// Mitsubishi GX Works2 project: Automation_EX2)   PLC: FX3G

// global labels: Global1
VAR_GLOBAL
  Start AT X007 : BOOL;
  Emergency AT X005 : BOOL;
  InventoryCheck AT M11 : BOOL;
  Valid AT M10 : BOOL;
  ReadyForWork AT Y007 : BOOL;
  IceCream AT X001 : BOOL;
  OpeningInventoryRaspberry AT D1100 : REAL;
  CurentInventoryRaspberry AT D1102 : REAL;
  OpeningInventoryLemon AT D1104 : REAL;
  CurentInventoryLemon AT D1106 : REAL;
  OpeningInventoryStabilizer AT D1108 : REAL;
  CurentInventoryStabilizer AT D1110 : REAL;
  OpeningInventoryGumy AT D1112 : REAL;
  CurentInventoryGumy AT D1114 : REAL;
  AnalogicInput AT D8280 : INT;
END_VAR
VAR_GLOBAL CONSTANT
  small5 : INT := 5;
  Big6 : INT := 6;
  Rgular : INT;
  Rgular5 : INT := 5;
  Rgular0 : INT;
  Treat6 : INT := 6;
  Treat10 : INT := 10;
END_VAR
VAR_GLOBAL
  Select_Regular AT M21 : BOOL;
  Select_Treat AT M31 : BOOL;
  SystemActive AT X007 : BOOL;
  Regular_Selected AT M100 : BOOL;
  Treat_Selected AT M200 : BOOL;
  Working_Lamp AT Y000 : BOOL;
  TC_5 AT TC5 : BOOL;
  Timer5_Done AT TS5 : BOOL;
END_VAR
VAR_GLOBAL CONSTANT
  Const_RR : REAL;
  Const_385 : REAL := 385.0;
  Const_210 : REAL := 210.0;
  Const_665 : REAL := 665.0;
  Const_70 : REAL := 70.0;
  Const_280 : REAL := 280.0;
  Const_105 : REAL := 105.0;
  Const_28 : REAL := 28.0;
  Const_455 : REAL := 455.0;
  Const_50 : INT := K50;
END_VAR
VAR_GLOBAL
  Timer5 AT TC50 : BOOL;
  CON50 AT K50 : INT;
  TC5 AT TC5 : BOOL;
  Timerrr AT TC5 : BOOL;
  Timer2 AT TC6 : BOOL;
  Timer2_done AT TS6 : BOOL;
  Shake AT X002 : BOOL;
  Cooling AT X002 : BOOL;
  Temp AT X003 : BOOL;
  CoolingTimer AT TC80 : BOOL;
  CON_80 AT K80 : INT;
  StageOneFinished AT M300 : BOOL;
  TempLowerThen10 AT X003 : BOOL;
  CoolTimerStop AT TC3 : BOOL;
  CoolTimerStoped AT TS80 : BOOL;
  CoolingLamp AT Y002 : BOOL;
  ReadyForShake AT M350 : BOOL;
END_VAR
VAR_GLOBAL CONSTANT
  Const280 : REAL := 280.0;
  Const_490 : REAL := 490.0;
END_VAR
VAR_GLOBAL
  LemonMakingTank AT D1116 : REAL;
  RaspberyMakingTank AT D1118 : REAL;
END_VAR
VAR_GLOBAL CONSTANT
  Const_350 : REAL := 350.0;
  Const_560 : REAL := 560.0;
  Const_700 : REAL := 700.0;
END_VAR
VAR_GLOBAL
  LemonCoolingTank AT D1120 : REAL;
  RaspberyCoolingTank AT D1122 : REAL;
  ShakingTank AT D1124 : REAL;
END_VAR
VAR_GLOBAL CONSTANT
  Const_1 : REAL := 1;
END_VAR
VAR_GLOBAL
  XXXXX AT M500 : BOOL;
  XXXXxx AT M500 : BOOL;
  Start_Mixing AT M500 : BOOL;
  Con30 AT K30 : INT;
  Mixing_Lamp AT TC30 : BOOL;
  Mixing_Reg_Lamp AT TC30 : BOOL;
  Mixing_Trt_Lamp AT TC50 : BOOL;
  Mixing_Done AT M501 : BOOL;
  Un_Timer AT TC21 : BOOL;
  Timer20 AT TS20 : BOOL;
  Timer21 AT TS21 : BOOL;
  Timer_20 AT TC20 : BOOL;
  Mixing_Lamp1 AT Y005 : BOOL;
  Mixing_Lamp2 AT Y006 : BOOL;
  Total_Packages AT D5000 : INT;
  M50Mixing_Done1 AT M501 : BOOL;
END_VAR
VAR_GLOBAL CONSTANT
  Rgular2000 : INT := 2000;
  Treat2400 : INT := 2400;
  Treat4000 : INT := 4000;
END_VAR
VAR_GLOBAL
  InventoryCheck12 AT M12 : BOOL;
  InventoryCheck13 AT M13 : BOOL;
  InventoryCheck14 AT M14 : BOOL;
  InventoryCheck15 AT M15 : BOOL;
  InventoryCheck16 AT M16 : BOOL;
  InventoryCheck17 AT M17 : BOOL;
  InventoryCheck18 AT M18 : BOOL;
  InventoryCheck19 AT M19 : BOOL;
  ReadyForShake1 AT M350 : BOOL;
  Start_Mixing1 AT M360 : BOOL;
  Mixing_Done1 AT M370 : BOOL;
  Station_Pack1 AT D5002 : REAL;
  Const10 AT E10 : REAL;
  Const_0 AT K0 : INT;
  Const_40 AT E40 : REAL;
  AnalogOutput AT D8282 : INT;
  Sensor_Error_Lamp AT Y011 : BOOL;
  Special_Relay AT M8013 : BOOL;
  Blink_Counter AT CS0 : BOOL;
  Const_5 AT K5 : INT;
  Analog_In_Error AT M380 : BOOL;
END_VAR
VAR_GLOBAL CONSTANT
  Treat4030 : INT := 4030;
  Rgular2030 : INT := 2030;
END_VAR
VAR_GLOBAL
  Low_Range_Regular AT M20 : BOOL;
  Low_Range_Treat AT M30 : BOOL;
END_VAR

// task Task_01 (event TRUE, interval 0, priority 31): POU_01

PROGRAM POU_01
(* structured ladder/FBD written out as ST: instructions are called as NAME(EN, inputs, outputs); _pN, _eN, _tN stand for wires *)
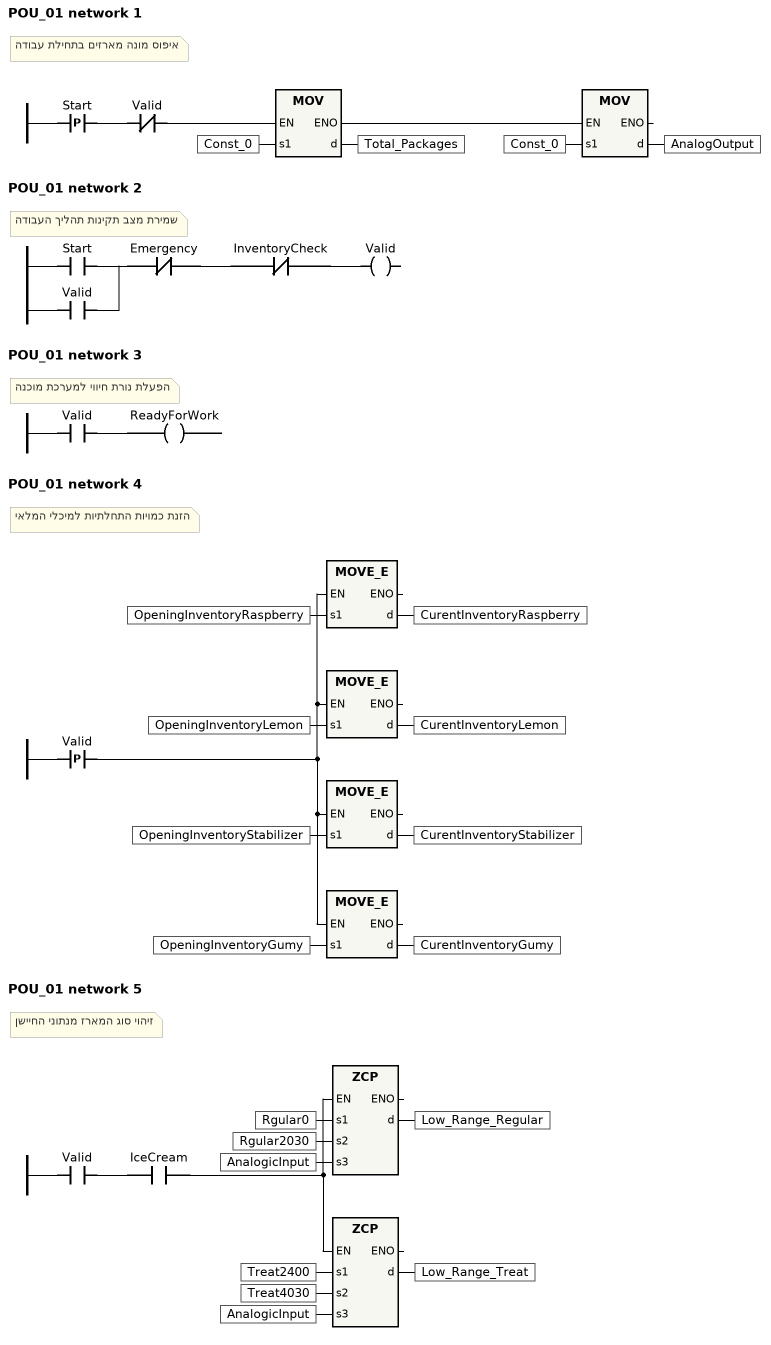
(* network 1 *)
(* איפוס מונה מארזים בתחילת עבודה *)
_e1 := MOV(LDP(TRUE, Start) AND NOT Valid, Const_0, Total_Packages);
MOV(_e1, Const_0, AnalogOutput);
(* network 2 *)
(* שמירת מצב תקינות תהליך העבודה *)
Valid := ((Start OR Valid) AND NOT Emergency) AND NOT InventoryCheck;
(* network 3 *)
(* הפעלת נורת חיווי למערכת מוכנה *)
ReadyForWork := Valid;
(* network 4 *)
(* הזנת כמויות התחלתיות למיכלי המלאי *)
_p1 := LDP(TRUE, Valid);
MOVE_E(_p1, OpeningInventoryRaspberry, CurentInventoryRaspberry);
MOVE_E(_p1, OpeningInventoryLemon, CurentInventoryLemon);
MOVE_E(_p1, OpeningInventoryStabilizer, CurentInventoryStabilizer);
MOVE_E(_p1, OpeningInventoryGumy, CurentInventoryGumy);
(* network 5 *)
(* זיהוי סוג המארז מנתוני החיישן *)
_p1 := Valid AND IceCream;
ZCP(_p1, Rgular0, Rgular2030, AnalogicInput, Low_Range_Regular);
ZCP(_p1, Treat2400, Treat4030, AnalogicInput, Low_Range_Treat);
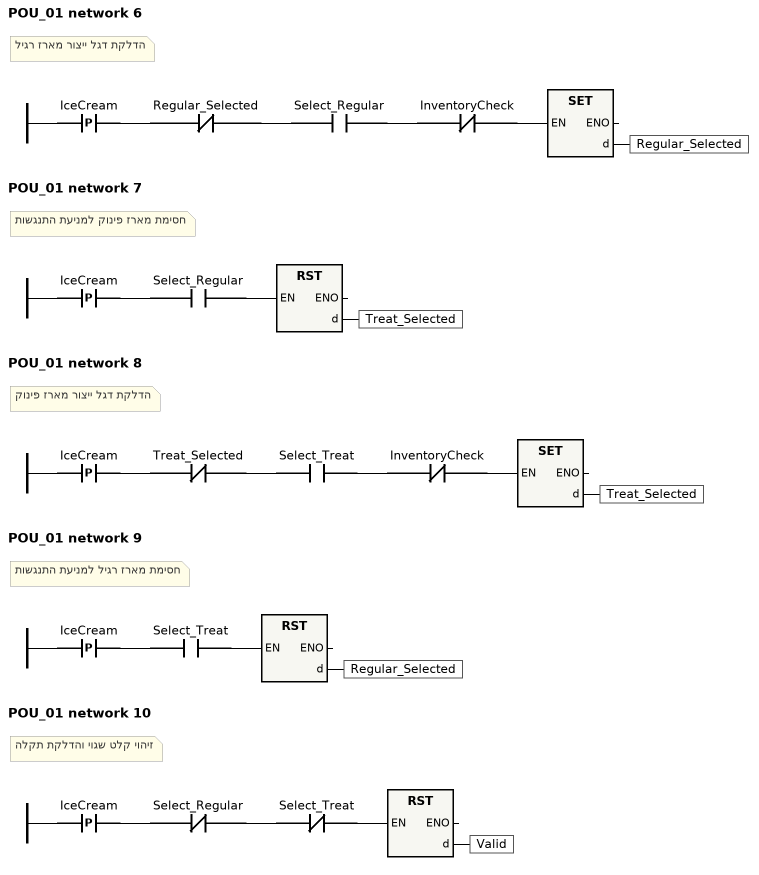
(* network 6 *)
(* הדלקת דגל ייצור מארז רגיל *)
SET(LDP(TRUE, IceCream) AND NOT Regular_Selected AND Select_Regular AND NOT InventoryCheck, Regular_Selected);
(* network 7 *)
(* חסימת מארז פינוק למניעת התנגשות *)
RST(LDP(TRUE, IceCream) AND Select_Regular, Treat_Selected);
(* network 8 *)
(* הדלקת דגל ייצור מארז פינוק *)
SET(LDP(TRUE, IceCream) AND NOT Treat_Selected AND Select_Treat AND NOT InventoryCheck, Treat_Selected);
(* network 9 *)
(* חסימת מארז רגיל למניעת התנגשות *)
RST(LDP(TRUE, IceCream) AND Select_Treat, Regular_Selected);
(* network 10 *)
(* זיהוי קלט שגוי והדלקת תקלה *)
RST(LDP(TRUE, IceCream) AND NOT Select_Regular AND NOT Select_Treat, Valid);
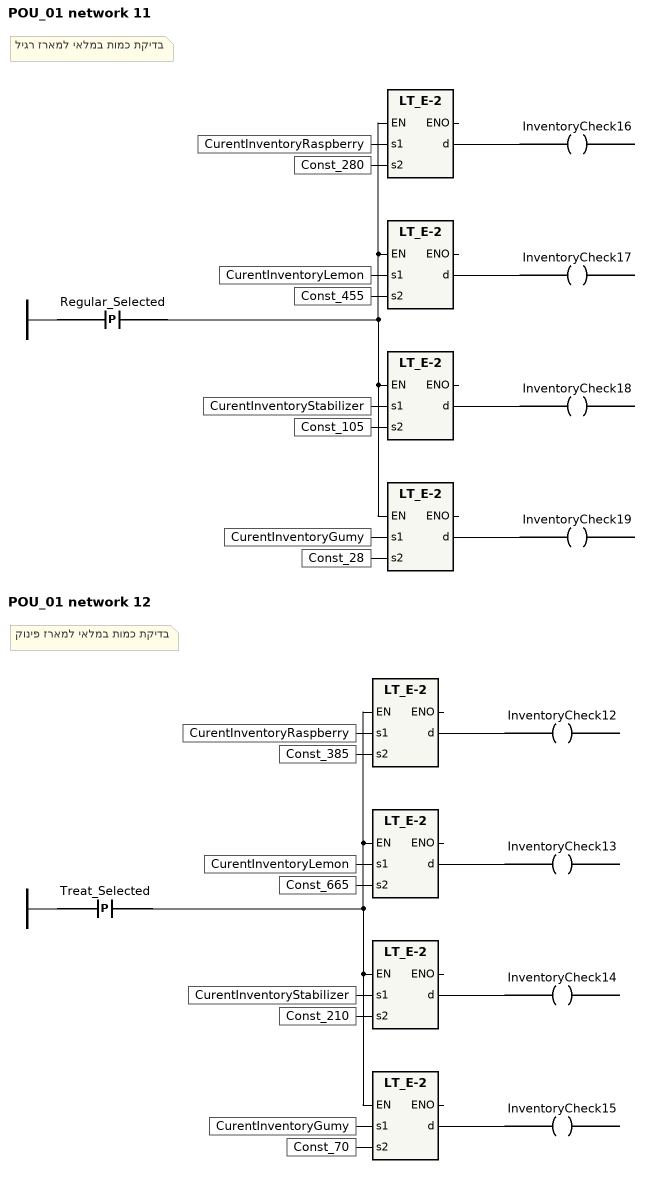
(* network 11 *)
(* בדיקת כמות במלאי למארז רגיל *)
_p1 := LDP(TRUE, Regular_Selected);
LT_E(_p1, CurentInventoryRaspberry, Const_280, _t2);
InventoryCheck16 := _t2;
LT_E(_p1, CurentInventoryLemon, Const_455, _t3);
InventoryCheck17 := _t3;
LT_E(_p1, CurentInventoryStabilizer, Const_105, _t4);
InventoryCheck18 := _t4;
LT_E(_p1, CurentInventoryGumy, Const_28, _t5);
InventoryCheck19 := _t5;
(* network 12 *)
(* בדיקת כמות במלאי למארז פינוק *)
_p1 := LDP(TRUE, Treat_Selected);
LT_E(_p1, CurentInventoryRaspberry, Const_385, _t2);
InventoryCheck12 := _t2;
LT_E(_p1, CurentInventoryLemon, Const_665, _t3);
InventoryCheck13 := _t3;
LT_E(_p1, CurentInventoryStabilizer, Const_210, _t4);
InventoryCheck14 := _t4;
LT_E(_p1, CurentInventoryGumy, Const_70, _t5);
InventoryCheck15 := _t5;
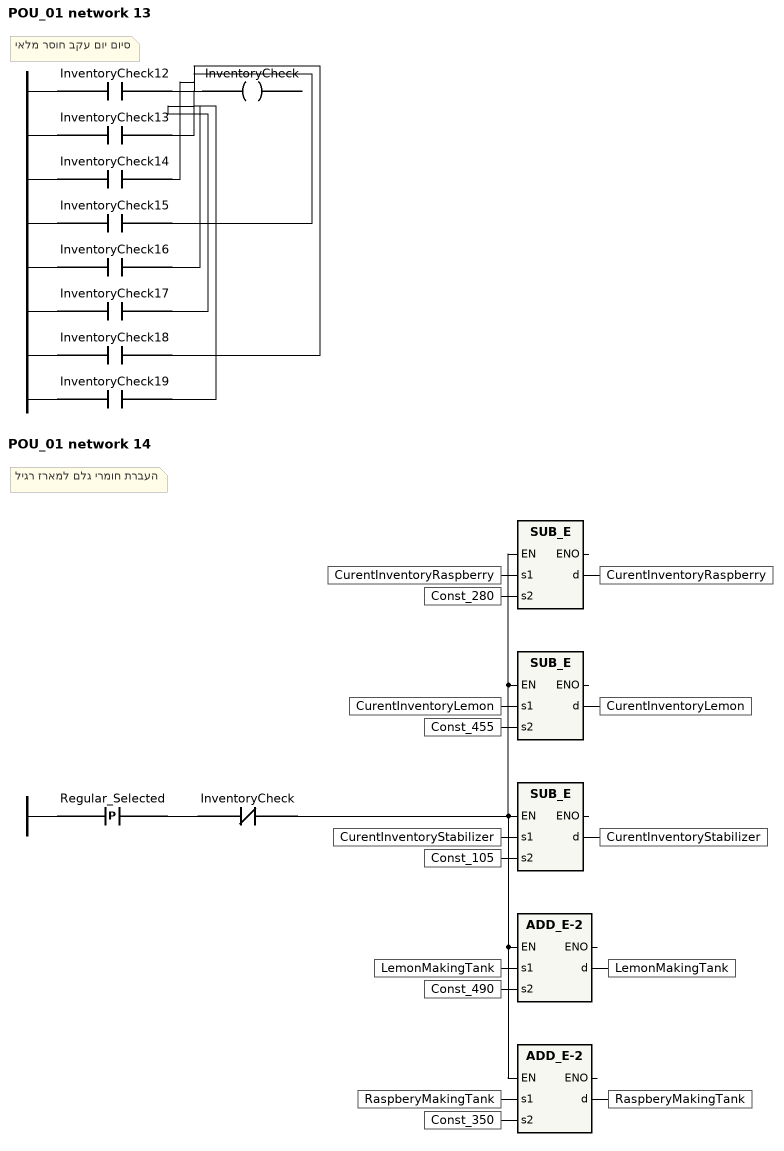
(* network 13 *)
(* סיום יום עקב חוסר מלאי *)
InventoryCheck := InventoryCheck12 OR InventoryCheck13 OR InventoryCheck14 OR InventoryCheck15 OR InventoryCheck16 OR InventoryCheck17 OR InventoryCheck18 OR InventoryCheck19;
(* network 14 *)
(* העברת חומרי גלם למארז רגיל *)
_p1 := LDP(TRUE, Regular_Selected) AND NOT InventoryCheck;
SUB_E(_p1, CurentInventoryRaspberry, Const_280, CurentInventoryRaspberry);
SUB_E(_p1, CurentInventoryLemon, Const_455, CurentInventoryLemon);
SUB_E(_p1, CurentInventoryStabilizer, Const_105, CurentInventoryStabilizer);
ADD_E(_p1, LemonMakingTank, Const_490, LemonMakingTank);
ADD_E(_p1, RaspberyMakingTank, Const_350, RaspberyMakingTank);
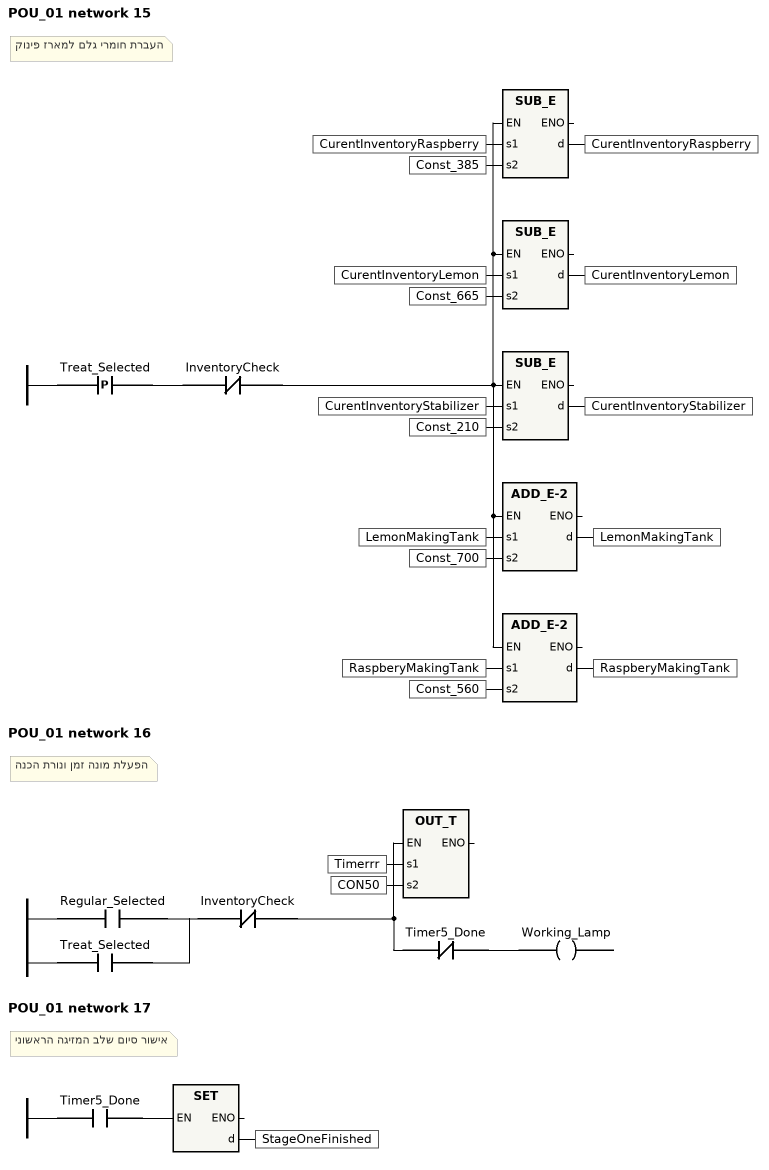
(* network 15 *)
(* העברת חומרי גלם למארז פינוק *)
_p1 := LDP(TRUE, Treat_Selected) AND NOT InventoryCheck;
SUB_E(_p1, CurentInventoryRaspberry, Const_385, CurentInventoryRaspberry);
SUB_E(_p1, CurentInventoryLemon, Const_665, CurentInventoryLemon);
SUB_E(_p1, CurentInventoryStabilizer, Const_210, CurentInventoryStabilizer);
ADD_E(_p1, LemonMakingTank, Const_700, LemonMakingTank);
ADD_E(_p1, RaspberyMakingTank, Const_560, RaspberyMakingTank);
(* network 16 *)
(* הפעלת מונה זמן ונורת הכנה *)
_p1 := (Regular_Selected OR Treat_Selected) AND NOT InventoryCheck;
OUT_T(_p1, Timerrr, CON50);
Working_Lamp := _p1 AND NOT Timer5_Done;
(* network 17 *)
(* אישור סיום שלב המזיגה הראשוני *)
SET(Timer5_Done, StageOneFinished);
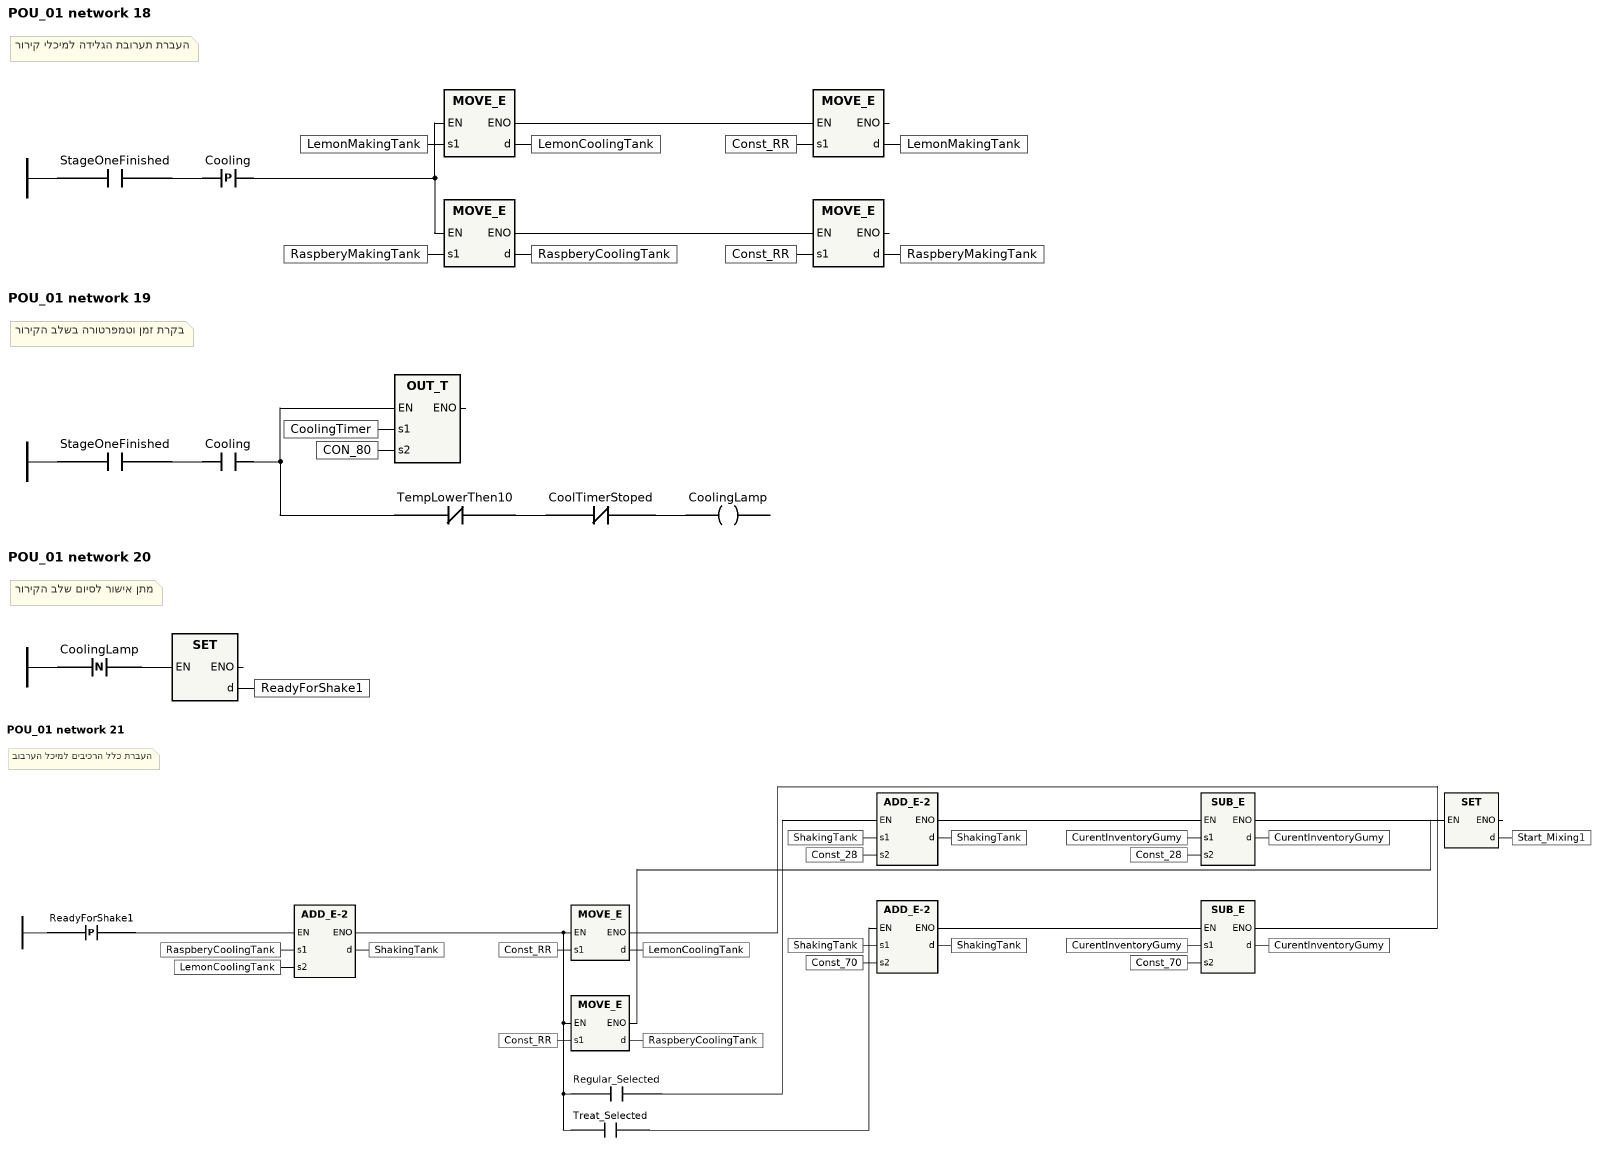
(* network 18 *)
(* העברת תערובת הגלידה למיכלי קירור *)
_p1 := StageOneFinished AND LDP(TRUE, Cooling);
_e2 := MOVE_E(_p1, LemonMakingTank, LemonCoolingTank);
MOVE_E(_e2, Const_RR, LemonMakingTank);
_e3 := MOVE_E(_p1, RaspberyMakingTank, RaspberyCoolingTank);
MOVE_E(_e3, Const_RR, RaspberyMakingTank);
(* network 19 *)
(* בקרת זמן וטמפרטורה בשלב הקירור *)
_p1 := StageOneFinished AND Cooling;
OUT_T(_p1, CoolingTimer, CON_80);
CoolingLamp := _p1 AND NOT TempLowerThen10 AND NOT CoolTimerStoped;
(* network 20 *)
(* מתן אישור לסיום שלב הקירור *)
SET(LDF(TRUE, CoolingLamp), ReadyForShake1);
(* network 21 *)
(* העברת כלל הרכיבים למיכל הערבוב *)
_e1 := ADD_E(LDP(TRUE, ReadyForShake1), RaspberyCoolingTank, LemonCoolingTank, ShakingTank);
_e2 := ADD_E(_e1 AND Regular_Selected, ShakingTank, Const_28, ShakingTank);
_e3 := SUB_E(_e2, CurentInventoryGumy, Const_28, CurentInventoryGumy);
_e4 := ADD_E(_e1 AND Treat_Selected, ShakingTank, Const_70, ShakingTank);
_e5 := SUB_E(_e4, CurentInventoryGumy, Const_70, CurentInventoryGumy);
_e6 := MOVE_E(_e1, Const_RR, LemonCoolingTank);
_e7 := MOVE_E(_e1, Const_RR, RaspberyCoolingTank);
SET(_e3 OR _e5 OR _e6 OR _e7, Start_Mixing1);
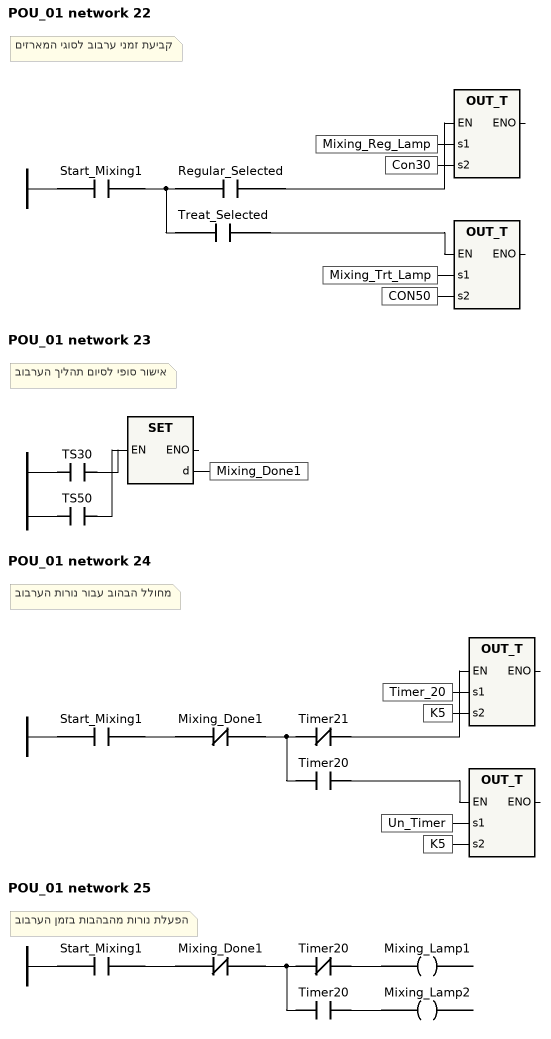
(* network 22 *)
(* קביעת זמני ערבוב לסוגי המארזים *)
OUT_T(Start_Mixing1 AND Regular_Selected, Mixing_Reg_Lamp, Con30);
OUT_T(Start_Mixing1 AND Treat_Selected, Mixing_Trt_Lamp, CON50);
(* network 23 *)
(* אישור סופי לסיום תהליך הערבוב *)
SET(TS30 OR TS50, Mixing_Done1);
(* network 24 *)
(* מחולל הבהוב עבור נורות הערבוב *)
_p1 := Start_Mixing1 AND NOT Mixing_Done1;
OUT_T(_p1 AND NOT Timer21, Timer_20, K5);
OUT_T(_p1 AND Timer20, Un_Timer, K5);
(* network 25 *)
(* הפעלת נורות מהבהבות בזמן הערבוב *)
_p1 := Start_Mixing1 AND NOT Mixing_Done1;
Mixing_Lamp1 := _p1 AND NOT Timer20;
Mixing_Lamp2 := _p1 AND Timer20;
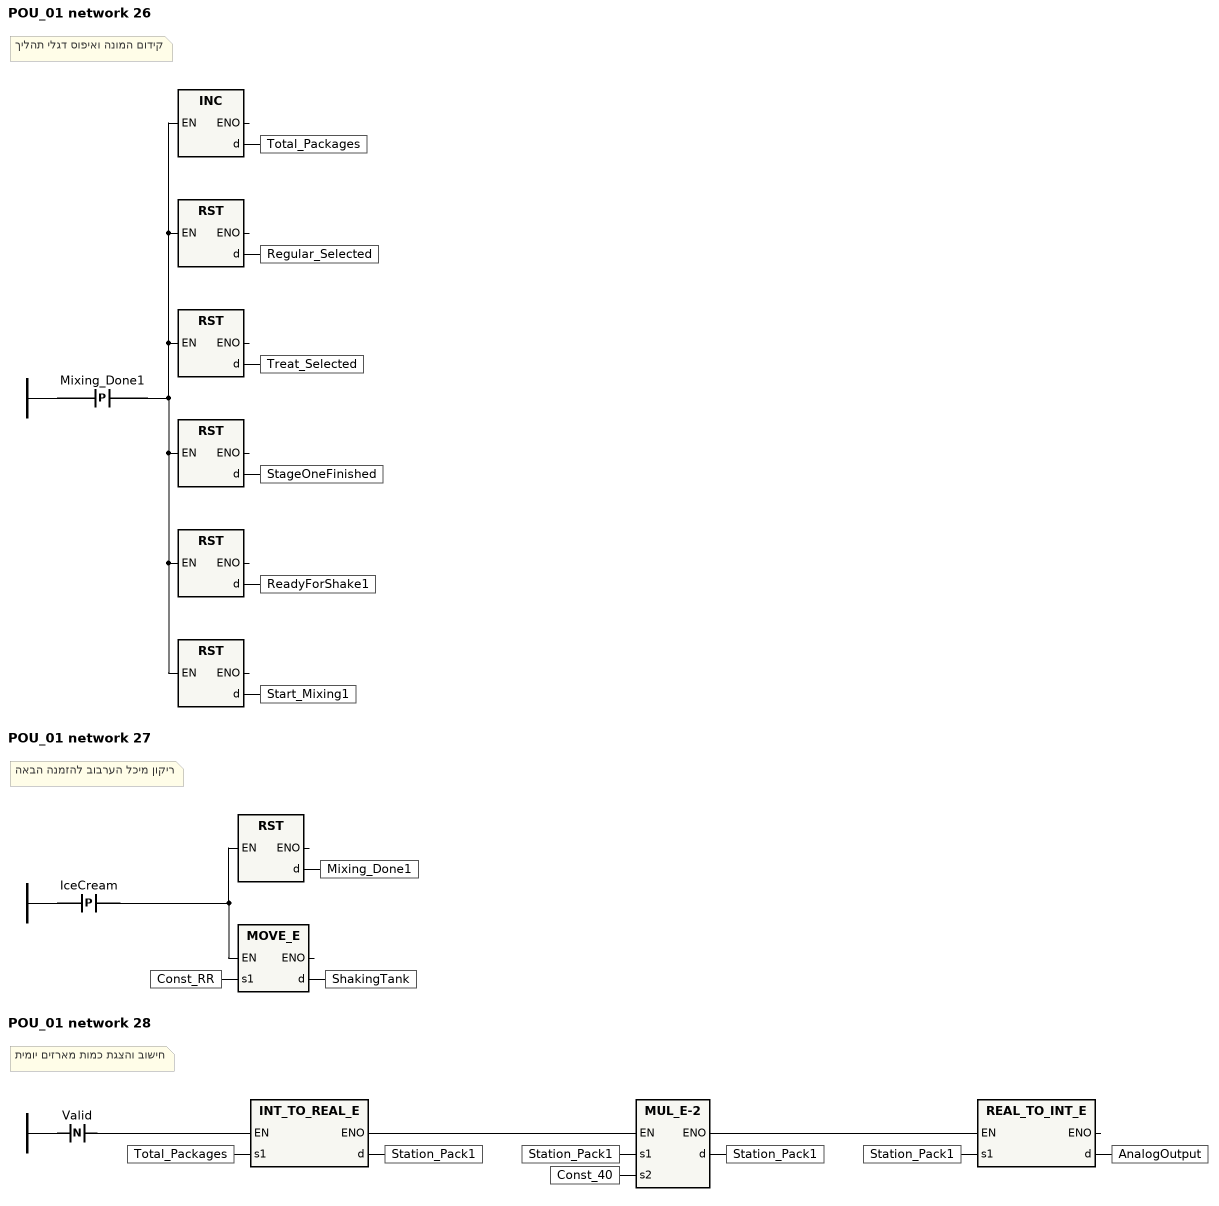
(* network 26 *)
(* קידום המונה ואיפוס דגלי תהליך *)
_p1 := LDP(TRUE, Mixing_Done1);
INC(_p1, Total_Packages);
RST(_p1, Regular_Selected);
RST(_p1, Treat_Selected);
RST(_p1, StageOneFinished);
RST(_p1, ReadyForShake1);
RST(_p1, Start_Mixing1);
(* network 27 *)
(* ריקון מיכל הערבוב להזמנה הבאה *)
_p1 := LDP(TRUE, IceCream);
RST(_p1, Mixing_Done1);
MOVE_E(_p1, Const_RR, ShakingTank);
(* network 28 *)
(* חישוב והצגת כמות מארזים יומית *)
_e1 := INT_TO_REAL_E(LDF(TRUE, Valid), Total_Packages, Station_Pack1);
_e2 := MUL_E(_e1, Station_Pack1, Const_40, Station_Pack1);
REAL_TO_INT_E(_e2, Station_Pack1, AnalogOutput);
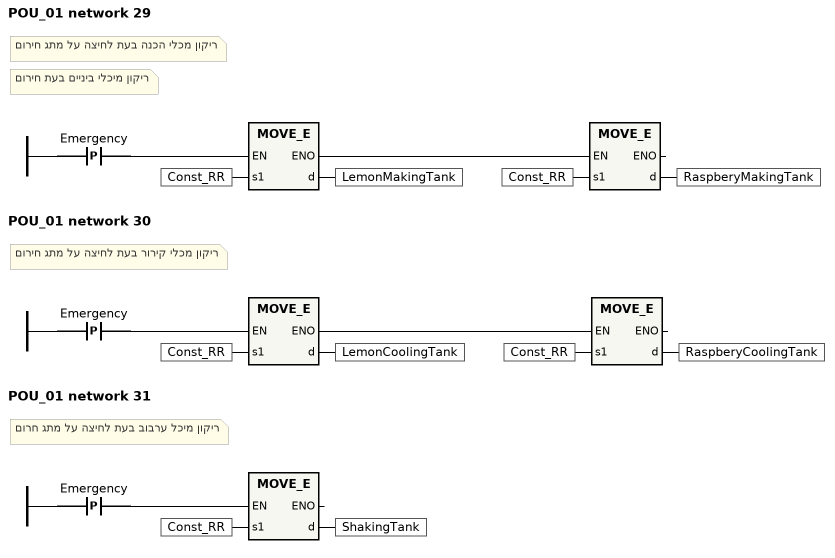
(* network 29 *)
(* ריקון מכלי הכנה בעת לחיצה על מתג חירום *)
(* ריקון מיכלי ביניים בעת חירום *)
_e1 := MOVE_E(LDP(TRUE, Emergency), Const_RR, LemonMakingTank);
MOVE_E(_e1, Const_RR, RaspberyMakingTank);
(* network 30 *)
(* ריקון מכלי קירור בעת לחיצה על מתג חירום *)
_e1 := MOVE_E(LDP(TRUE, Emergency), Const_RR, LemonCoolingTank);
MOVE_E(_e1, Const_RR, RaspberyCoolingTank);
(* network 31 *)
(* ריקון מיכל ערבוב בעת לחיצה על מתג חרום *)
MOVE_E(LDP(TRUE, Emergency), Const_RR, ShakingTank);
END_PROGRAM

// device comments not shown above
D1100  ; OpeningInventoryRaspberry
D1102  ; OpeningInventoryLemon
D1104  ; OpeningInventoryStabilizer
D1106  ; OpeningInventoryGumy
D1110  ; CurentInventoryRaspberry
D1112  ; CurentInventoryLemon
D1114  ; CurentInventoryStabilizer
D1116  ; CurentInventoryGumy
